PROGRAM PRG_CML_02_LoweratorCtrl
VAR
	tofRotaryDwell				: TOF;
	rtigTransferInHome		: R_TRIG;
	rtigTransferOnInit			: R_TRIG;
	rsRotaryHomeReq			: RS;
	rsRotaryRun				: RS;

	rtrigLoweratorInitByCP		: R_TRIG;
	tofLoweratorConvTimeOut	: FB_TOFR;
	tofLoweratorConvDelay	: TOF;

	tofRejectConvDelay		: FB_TOFR;

END_VAR

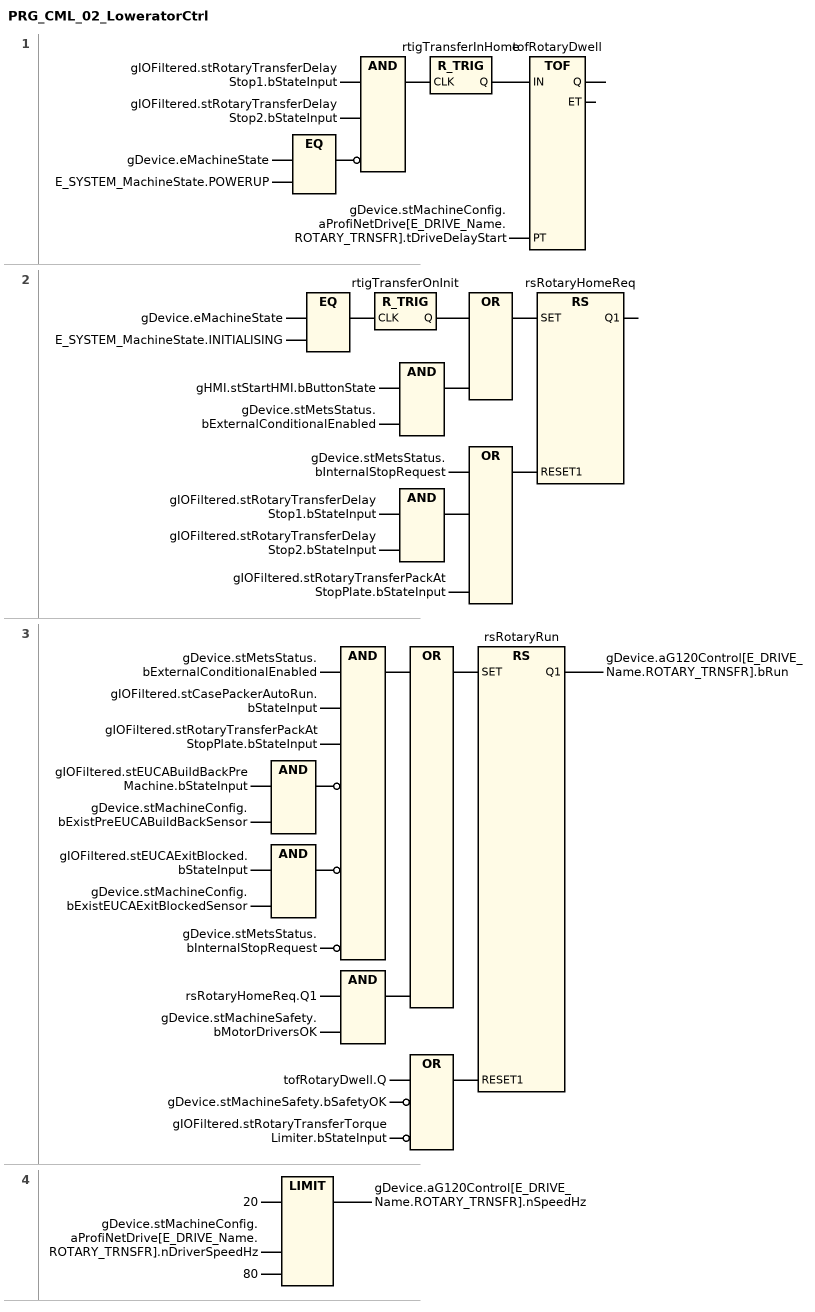
// NETWORK 1
rtigTransferInHome(CLK := gIOFiltered.stRotaryTransferDelayStop1.bStateInput AND gIOFiltered.stRotaryTransferDelayStop2.bStateInput AND NOT (gDevice.eMachineState = E_SYSTEM_MachineState.POWERUP)); // R_TRIG
tofRotaryDwell(IN := rtigTransferInHome.Q, PT := gDevice.stMachineConfig.aProfiNetDrive[E_DRIVE_Name.ROTARY_TRNSFR].tDriveDelayStart); // TOF

// NETWORK 2
rtigTransferOnInit(CLK := gDevice.eMachineState = E_SYSTEM_MachineState.INITIALISING); // R_TRIG
rsRotaryHomeReq(SET := rtigTransferOnInit.Q OR gHMI.stStartHMI.bButtonState AND gDevice.stMetsStatus.bExternalConditionalEnabled, RESET1 := gDevice.stMetsStatus.bInternalStopRequest OR gIOFiltered.stRotaryTransferDelayStop1.bStateInput AND gIOFiltered.stRotaryTransferDelayStop2.bStateInput OR gIOFiltered.stRotaryTransferPackAtStopPlate.bStateInput); // RS

// NETWORK 3
rsRotaryRun(SET := gDevice.stMetsStatus.bExternalConditionalEnabled AND gIOFiltered.stCasePackerAutoRun.bStateInput AND gIOFiltered.stRotaryTransferPackAtStopPlate.bStateInput AND NOT (gIOFiltered.stEUCABuildBackPreMachine.bStateInput AND gDevice.stMachineConfig.bExistPreEUCABuildBackSensor) AND NOT (gIOFiltered.stEUCAExitBlocked.bStateInput AND gDevice.stMachineConfig.bExistEUCAExitBlockedSensor) AND NOT gDevice.stMetsStatus.bInternalStopRequest OR rsRotaryHomeReq.Q1 AND gDevice.stMachineSafety.bMotorDriversOK, RESET1 := tofRotaryDwell.Q OR NOT gDevice.stMachineSafety.bSafetyOK OR NOT gIOFiltered.stRotaryTransferTorqueLimiter.bStateInput); // RS
gDevice.aG120Control[E_DRIVE_Name.ROTARY_TRNSFR].bRun := rsRotaryRun.Q1;

// NETWORK 4
gDevice.aG120Control[E_DRIVE_Name.ROTARY_TRNSFR].nSpeedHz := LIMIT(20, gDevice.stMachineConfig.aProfiNetDrive[E_DRIVE_Name.ROTARY_TRNSFR].nDriverSpeedHz, 80);

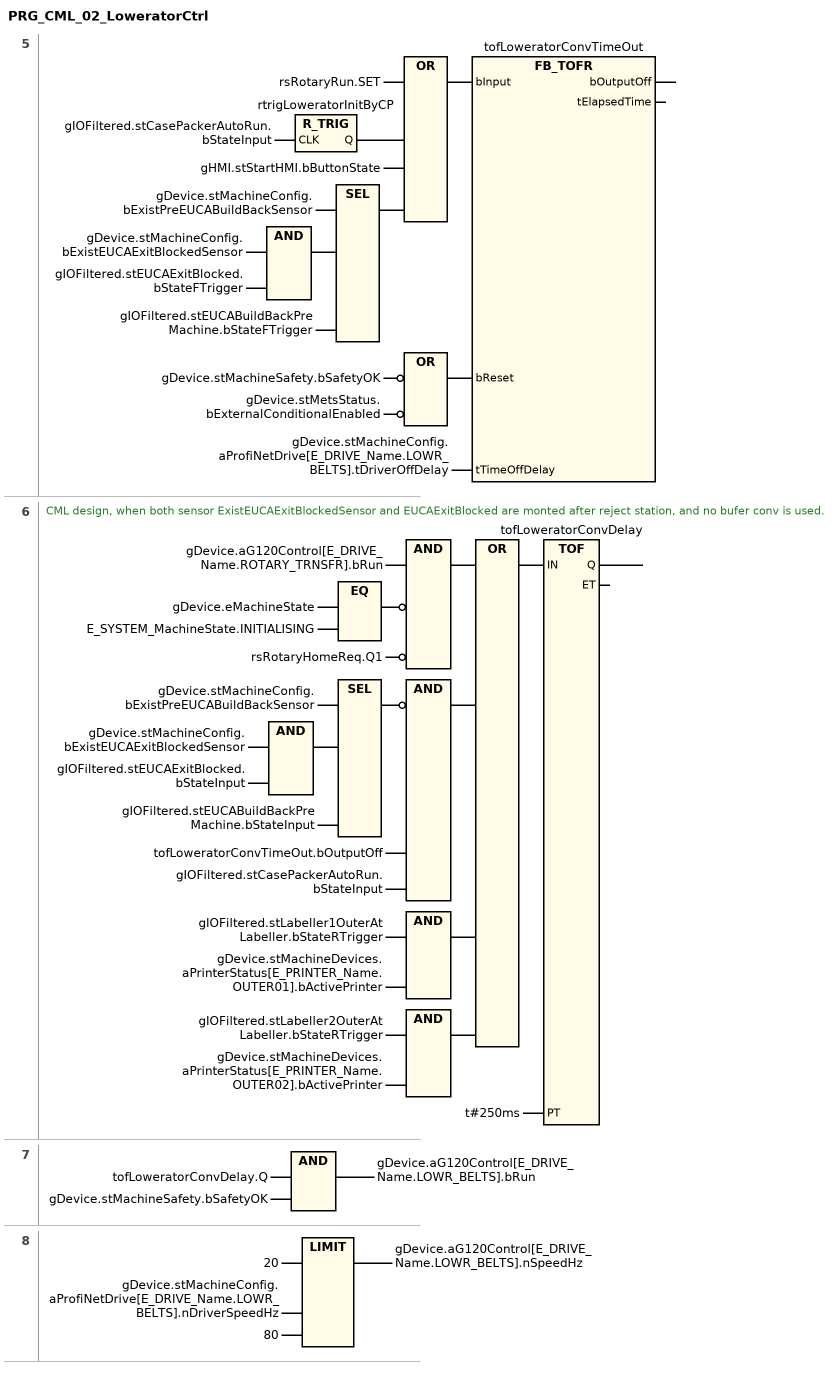
// NETWORK 5
rtrigLoweratorInitByCP(CLK := gIOFiltered.stCasePackerAutoRun.bStateInput); // R_TRIG
tofLoweratorConvTimeOut(
    bInput := rsRotaryRun.SET OR rtrigLoweratorInitByCP.Q OR gHMI.stStartHMI.bButtonState OR SEL(gDevice.stMachineConfig.bExistPreEUCABuildBackSensor, gDevice.stMachineConfig.bExistEUCAExitBlockedSensor AND gIOFiltered.stEUCAExitBlocked.bStateFTrigger, gIOFiltered.stEUCABuildBackPreMachine.bStateFTrigger),
    bReset := NOT gDevice.stMachineSafety.bSafetyOK OR NOT gDevice.stMetsStatus.bExternalConditionalEnabled,
    tTimeOffDelay := gDevice.stMachineConfig.aProfiNetDrive[E_DRIVE_Name.LOWR_BELTS].tDriverOffDelay); // FB_TOFR

// NETWORK 6
// CML design, when both sensor ExistEUCAExitBlockedSensor and EUCAExitBlocked are monted after reject station, and no bufer conv is used.
tofLoweratorConvDelay(IN := gDevice.aG120Control[E_DRIVE_Name.ROTARY_TRNSFR].bRun AND NOT (gDevice.eMachineState = E_SYSTEM_MachineState.INITIALISING) AND NOT rsRotaryHomeReq.Q1 OR NOT SEL(gDevice.stMachineConfig.bExistPreEUCABuildBackSensor, gDevice.stMachineConfig.bExistEUCAExitBlockedSensor AND gIOFiltered.stEUCAExitBlocked.bStateInput, gIOFiltered.stEUCABuildBackPreMachine.bStateInput) AND tofLoweratorConvTimeOut.bOutputOff AND gIOFiltered.stCasePackerAutoRun.bStateInput OR gIOFiltered.stLabeller1OuterAtLabeller.bStateRTrigger AND gDevice.stMachineDevices.aPrinterStatus[E_PRINTER_Name.OUTER01].bActivePrinter OR gIOFiltered.stLabeller2OuterAtLabeller.bStateRTrigger AND gDevice.stMachineDevices.aPrinterStatus[E_PRINTER_Name.OUTER02].bActivePrinter, PT := t#250ms); // TOF

// NETWORK 7
gDevice.aG120Control[E_DRIVE_Name.LOWR_BELTS].bRun := tofLoweratorConvDelay.Q AND gDevice.stMachineSafety.bSafetyOK;

// NETWORK 8
gDevice.aG120Control[E_DRIVE_Name.LOWR_BELTS].nSpeedHz := LIMIT(20, gDevice.stMachineConfig.aProfiNetDrive[E_DRIVE_Name.LOWR_BELTS].nDriverSpeedHz, 80);

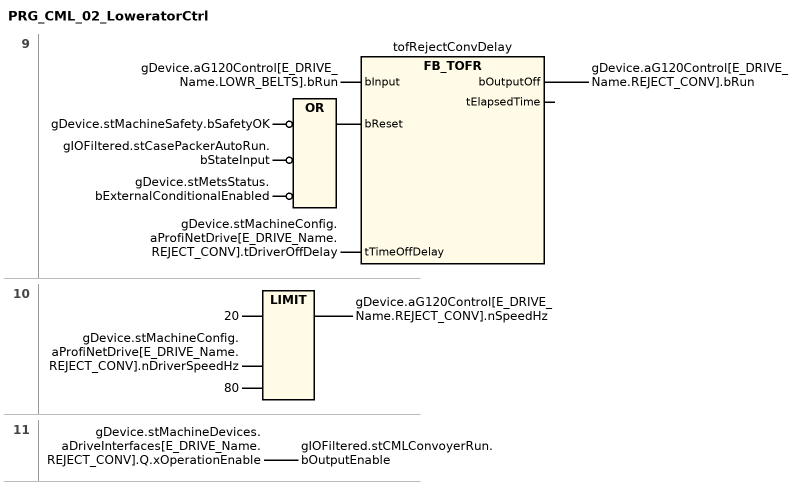
// NETWORK 9
tofRejectConvDelay(
    bInput := gDevice.aG120Control[E_DRIVE_Name.LOWR_BELTS].bRun,
    bReset := NOT gDevice.stMachineSafety.bSafetyOK OR NOT gIOFiltered.stCasePackerAutoRun.bStateInput OR NOT gDevice.stMetsStatus.bExternalConditionalEnabled,
    tTimeOffDelay := gDevice.stMachineConfig.aProfiNetDrive[E_DRIVE_Name.REJECT_CONV].tDriverOffDelay); // FB_TOFR
gDevice.aG120Control[E_DRIVE_Name.REJECT_CONV].bRun := tofRejectConvDelay.bOutputOff;

// NETWORK 10
gDevice.aG120Control[E_DRIVE_Name.REJECT_CONV].nSpeedHz := LIMIT(20, gDevice.stMachineConfig.aProfiNetDrive[E_DRIVE_Name.REJECT_CONV].nDriverSpeedHz, 80);

// NETWORK 11
gIOFiltered.stCMLConvoyerRun.bOutputEnable := gDevice.stMachineDevices.aDriveInterfaces[E_DRIVE_Name.REJECT_CONV].Q.xOperationEnable;

END_PROGRAM

(* stored: Version 1.1.0.1
   POU PRG_CML_02_LoweratorCtrl: Id {c5c5cbd4-6c96-4e4d-9dd4-072f0906d65f}, SpecialFunc None *)
